TYPE ST_DebugSensors_TransferUnitEmulation :
STRUCT
	EnableSensorDebug	: BOOL; 					// Overwrite sensor values with debug sensor values
	HW_Inputs			: ST_HW_InputsTransferUnit;	// Debug sensors
END_STRUCT
END_TYPE

(* stored: Version 1.1.0.1, ProductVersion 3.1.4024.9
   DUT ST_DebugSensors_TransferUnitEmulation: Id {9f01885c-6a75-41fe-b4c7-ff20500dcd9c} *)
